FUNCTION_BLOCK Hutschienenmoped_XL_8_DO_PWM (* Service Interface Function Block Type *)
  (* Function: All Outputs; Description: this maps to QX this is a Digital Out with a Soft Start and a DutyCycle. this is SoftStart only, the Stop will be hard (e.g. to utilize like Stop on a Stop Switch) *)
  (* Version 1.0, 2018-12-05, Jose Cabral *)
  (* Version 1.1, 2022-08-04, Franz Höpfinger, HR Agrartechnik GmbH *)
  (* Version 1.2, 2023-01-05, Franz Höpfinger, HR Agrartechnik GmbH *)
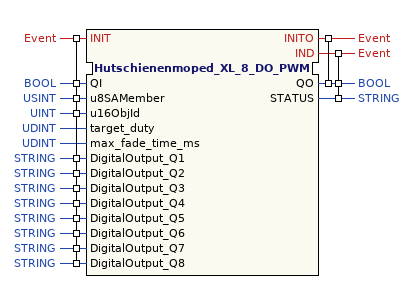
  EVENT_INPUT
    INIT WITH QI, u8SAMember, u16ObjId, DigitalOutput_Q1, DigitalOutput_Q2, DigitalOutput_Q3, DigitalOutput_Q4, DigitalOutput_Q5, DigitalOutput_Q6, DigitalOutput_Q7, DigitalOutput_Q8; (* Service Initialization *)
  END_EVENT
  EVENT_OUTPUT
    INITO WITH QO; (* Initialization Confirm *)
    IND WITH QO, STATUS; (* Indication from Resource *)
  END_EVENT
  VAR_INPUT
    QI : BOOL; (* Event Input Qualifier *)
    u8SAMember : USINT := GLOBAL; (* Dummy !, set to GLOBAL if in doubt. OFF deactivates FB. *)
    u16ObjId : UINT := ID_NULL; (* Dummy ! set to ID_NULL if in Doubt. ID_OFF deactivates FB. *)
    target_duty : UDINT;
    max_fade_time_ms : UDINT;
    DigitalOutput_Q1 : STRING;
    DigitalOutput_Q2 : STRING;
    DigitalOutput_Q3 : STRING;
    DigitalOutput_Q4 : STRING;
    DigitalOutput_Q5 : STRING;
    DigitalOutput_Q6 : STRING;
    DigitalOutput_Q7 : STRING;
    DigitalOutput_Q8 : STRING;
  END_VAR
  VAR_OUTPUT
    QO : BOOL; (* Event Output Qualifier *)
    STATUS : STRING; (* Service Status *)
  END_VAR
END_FUNCTION_BLOCK
